FUNCTION_BLOCK TestArrayVariables
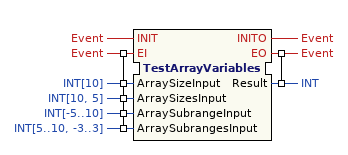
  EVENT_INPUT
    INIT;
    EI WITH ArraySizeInput, ArraySizesInput, ArraySubrangeInput, ArraySubrangesInput;
  END_EVENT
  EVENT_OUTPUT
    INITO;
    EO WITH Result;
  END_EVENT
  VAR_INPUT
    ArraySizeInput : ARRAY [0..9] OF INT;
    ArraySizesInput : ARRAY [10, 5] OF INT;
    ArraySubrangeInput : ARRAY [-5..10] OF INT;
    ArraySubrangesInput : ARRAY [5..10, -3..3] OF INT;
  END_VAR
  VAR_OUTPUT
    Result : INT;
  END_VAR
  EC_STATES
    START;
  END_STATES
  ALGORITHM TestAlg IN ST:
Result := ArraySizeInput[0] + ArraySizesInput[1, 2] + ArraySubrangeInput[-3] + ArraySubrangesInput[6, 0];&#38;#10;
  END_ALGORITHM
END_FUNCTION_BLOCK
